(*
    This function block is responsible for printing the results of the assertions using the built-in
    ADSLOGSTR functionality provided by the Tc2_System library. This sends the result using ADS, which
    is consumed by the error list of Visual Studio.
*)
FUNCTION_BLOCK FB_AdsAssertMessageFormatter IMPLEMENTS I_AssertMessageFormatter

METHOD PUBLIC LogAssertFailure
VAR_INPUT
    Expected : T_MaxString;
    Actual : T_MaxString;
    Message : T_MaxString;
    TestInstancePath : T_MaxString;
END_VAR
VAR
    AdjustAssertFailureMessageToMaxAllowedLength : FB_AdjustAssertFailureMessageToMaxAllowedLength;
    TestInstancePathCleaned : T_MaxString;
    TestInstancePathFinal : T_MaxString;
    ReturnValue : DINT;
    TestInstancePathProcessed : T_MaxString;
    MessagePart2 : T_MaxString;
    MessagePart3 : T_MaxString;
    MessagePart4 : T_MaxString;
    MessageProcessed : T_MaxString;
    Length2 : INT;
    Length3 : INT;
    Length4 : INT;
    LengthTotal : INT;
END_VAR
VAR CONSTANT
    MESSAGE_FORMATTED_STRING_MAX_NUMBER_OF_CHARACTERS : INT := 252; // The maximum printed text length is 250. The '%s' placeholder will be replaced, therefore the limit to use in the check is 252.
    ACTEXP_MAX_NUMBER_OF_CHARACTERS : INT := 250;
    TOO_LONG : STRING := '...too long';
END_VAR
TestInstancePathCleaned := F_RemoveInstancePathAndProjectNameFromTestInstancePath(TestInstancePath);
TestInstancePathFinal := CONCAT(STR1 := 'FAILED TEST $'',
                                STR2 := TestInstancePathCleaned);
TestInstancePathFinal := CONCAT(STR1 := TestInstancePathFinal,
                                STR2 := '$'');

MessagePart2 := CONCAT(STR1 := 'EXP: ',
                       STR2 := Expected);
MessagePart3 := CONCAT(STR1 := 'ACT: ',
                       STR2 := Actual);
IF LEN(STR := Message) > 0 THEN
    MessagePart4 := ', MSG: %s';
    Length4 := LEN(STR := MessagePart4)
             + LEN(STR := Message);
END_IF

IF (GVL_Param_TcUnit.MultipleLinesPerAssertionMessage) THEN
    Length2 := LEN(MessagePart2);
    IF (Length2 > ACTEXP_MAX_NUMBER_OF_CHARACTERS) THEN
        MessagePart2 := LEFT(STR := MessagePart2,
                             SIZE := ACTEXP_MAX_NUMBER_OF_CHARACTERS - LEN(STR := TOO_LONG));
        MessagePart2 := CONCAT (STR1 := MessagePart2,
                                STR2 := TOO_LONG);
        Length2 := LEN(MessagePart2);
    END_IF
    
    Length3 := LEN(MessagePart3);
    IF (Length3 > ACTEXP_MAX_NUMBER_OF_CHARACTERS) THEN
        MessagePart3 := LEFT(STR := MessagePart3,
                             SIZE := ACTEXP_MAX_NUMBER_OF_CHARACTERS - LEN(STR := TOO_LONG));
        MessagePart3 := CONCAT (STR1 := MessagePart3,
                                STR2 := TOO_LONG);
        Length3 := LEN(MessagePart3);
    END_IF

    LengthTotal := LEN(TestInstancePathFinal) + 2 + Length2 + 2 + Length3 + Length4;
END_IF

IF (LengthTotal <= MESSAGE_FORMATTED_STRING_MAX_NUMBER_OF_CHARACTERS) THEN
    // If the message must be printed on a single line ("multiple lines" disabled), then LengthTotal is not calculated, so this path is executed.
    TestInstancePathFinal := CONCAT(STR1 := TestInstancePathFinal,
                                    STR2 := ', ');
    TestInstancePathFinal := CONCAT(STR1 := TestInstancePathFinal,
                                    STR2 := MessagePart2);
    
    TestInstancePathFinal := CONCAT(STR1 := TestInstancePathFinal,
                                    STR2 := ', ');
    TestInstancePathFinal := CONCAT(STR1 := TestInstancePathFinal,
                                    STR2 := MessagePart3);
    
    IF Length4 > 0 THEN
        TestInstancePathFinal := CONCAT(STR1 := TestInstancePathFinal,
                                        STR2 := MessagePart4);
    END_IF
    
    AdjustAssertFailureMessageToMaxAllowedLength(TestInstancePath := TestInstancePathFinal,
                                                 TestMessage := Message,
                                                 TestInstancePathProcessed => TestInstancePathProcessed,
                                                 TestMessageProcessed => MessageProcessed);
    
    GVL_TcUnit.AdsMessageQueue.WriteLog(MsgCtrlMask := ADSLOG_MSGTYPE_ERROR,
                                        MsgFmtStr := TestInstancePathProcessed,
                                        StrArg := MessageProcessed);
    
// ELSE: print multiple lines
ELSIF (LEN(TestInstancePathFinal) + 2 + Length2 + 2 + Length3 <= MESSAGE_FORMATTED_STRING_MAX_NUMBER_OF_CHARACTERS) THEN
    // A message exists, because the text with message does not fit in one line, but it fits without the message. Print only the message in a separate line.
    TestInstancePathFinal := CONCAT(STR1 := TestInstancePathFinal,
                                    STR2 := ', ');
    TestInstancePathFinal := CONCAT(STR1 := TestInstancePathFinal,
                                    STR2 := MessagePart2);
    
    TestInstancePathFinal := CONCAT(STR1 := TestInstancePathFinal,
                                    STR2 := ', ');
    TestInstancePathFinal := CONCAT(STR1 := TestInstancePathFinal,
                                    STR2 := MessagePart3);
    
    AdjustAssertFailureMessageToMaxAllowedLength(TestInstancePath := TestInstancePathFinal,
                                                 TestMessage := '',
                                                 TestInstancePathProcessed => TestInstancePathProcessed,
                                                 TestMessageProcessed => MessageProcessed);
    
    GVL_TcUnit.AdsMessageQueue.WriteLog(MsgCtrlMask := ADSLOG_MSGTYPE_ERROR,
                                        MsgFmtStr := TestInstancePathProcessed,
                                        StrArg := MessageProcessed);
    
    // MessagePart4 (MSG)
    AdjustAssertFailureMessageToMaxAllowedLength(TestInstancePath := '_ MSG: %s',
                                                 TestMessage := Message,
                                                 TestInstancePathProcessed => TestInstancePathProcessed,
                                                 TestMessageProcessed => MessageProcessed);
    
    GVL_TcUnit.AdsMessageQueue.WriteLog(MsgCtrlMask := ADSLOG_MSGTYPE_ERROR,
                                        MsgFmtStr := TestInstancePathProcessed,
                                        StrArg := MessageProcessed);
    
ELSIF (2 + Length2 + 2 + Length3 <= ACTEXP_MAX_NUMBER_OF_CHARACTERS) THEN
    // Text without message does not fit in one line. EXP and ACT fit in one line, therefore print them together in 2nd line. Print message (if existing) in 3rd line.
    AdjustAssertFailureMessageToMaxAllowedLength(TestInstancePath := TestInstancePathFinal,
                                                 TestMessage := '',
                                                 TestInstancePathProcessed => TestInstancePathProcessed,
                                                 TestMessageProcessed => MessageProcessed);
    
    GVL_TcUnit.AdsMessageQueue.WriteLog(MsgCtrlMask := ADSLOG_MSGTYPE_ERROR,
                                        MsgFmtStr := TestInstancePathProcessed,
                                        StrArg := MessageProcessed);
    
    // MessagePart2 (EXP) + MessagePart3 (ACT)
    MessagePart2 := CONCAT (STR1 := '_ ',
                            STR2 := MessagePart2);
    MessagePart2 := CONCAT (STR1 := MessagePart2,
                            STR2 := ', ');
    MessagePart2 := CONCAT (STR1 := MessagePart2,
                            STR2 := MessagePart3);
    
    AdjustAssertFailureMessageToMaxAllowedLength(TestInstancePath := MessagePart2,
                                                 TestMessage := '',
                                                 TestInstancePathProcessed => TestInstancePathProcessed,
                                                 TestMessageProcessed => MessageProcessed);
    
    GVL_TcUnit.AdsMessageQueue.WriteLog(MsgCtrlMask := ADSLOG_MSGTYPE_ERROR,
                                        MsgFmtStr := TestInstancePathProcessed,
                                        StrArg := MessageProcessed);
    
    // MessagePart4 (MSG)
    IF Length4 > 0 THEN
        AdjustAssertFailureMessageToMaxAllowedLength(TestInstancePath := '_ MSG: %s',
                                                     TestMessage := Message,
                                                     TestInstancePathProcessed => TestInstancePathProcessed,
                                                     TestMessageProcessed => MessageProcessed);
        
        GVL_TcUnit.AdsMessageQueue.WriteLog(MsgCtrlMask := ADSLOG_MSGTYPE_ERROR,
                                            MsgFmtStr := TestInstancePathProcessed,
                                            StrArg := MessageProcessed);
    END_IF
ELSE
    // print every item in a separate line.
    AdjustAssertFailureMessageToMaxAllowedLength(TestInstancePath := TestInstancePathFinal,
                                                 TestMessage := '',
                                                 TestInstancePathProcessed => TestInstancePathProcessed,
                                                 TestMessageProcessed => MessageProcessed);
    
    GVL_TcUnit.AdsMessageQueue.WriteLog(MsgCtrlMask := ADSLOG_MSGTYPE_ERROR,
                                        MsgFmtStr := TestInstancePathProcessed,
                                        StrArg := MessageProcessed);
    
    // MessagePart2 (EXP)
    MessagePart2 := CONCAT (STR1 := '_ ',
                            STR2 := MessagePart2);

    AdjustAssertFailureMessageToMaxAllowedLength(TestInstancePath := MessagePart2,
                                                 TestMessage := '',
                                                 TestInstancePathProcessed => TestInstancePathProcessed,
                                                 TestMessageProcessed => MessageProcessed);
    
    GVL_TcUnit.AdsMessageQueue.WriteLog(MsgCtrlMask := ADSLOG_MSGTYPE_ERROR,
                                        MsgFmtStr := TestInstancePathProcessed,
                                        StrArg := MessageProcessed);
    
    // MessagePart3 (ACT)
    MessagePart3 := CONCAT (STR1 := '_ ',
                            STR2 := MessagePart3);
    
    AdjustAssertFailureMessageToMaxAllowedLength(TestInstancePath := MessagePart3,
                                                 TestMessage := '',
                                                 TestInstancePathProcessed => TestInstancePathProcessed,
                                                 TestMessageProcessed => MessageProcessed);
    
    GVL_TcUnit.AdsMessageQueue.WriteLog(MsgCtrlMask := ADSLOG_MSGTYPE_ERROR,
                                        MsgFmtStr := TestInstancePathProcessed,
                                        StrArg := MessageProcessed);
    
    // MessagePart4 (MSG)
    IF Length4 > 0 THEN
        AdjustAssertFailureMessageToMaxAllowedLength(TestInstancePath := '_ MSG: %s',
                                                     TestMessage := Message,
                                                     TestInstancePathProcessed => TestInstancePathProcessed,
                                                     TestMessageProcessed => MessageProcessed);
        
        GVL_TcUnit.AdsMessageQueue.WriteLog(MsgCtrlMask := ADSLOG_MSGTYPE_ERROR,
                                            MsgFmtStr := TestInstancePathProcessed,
                                            StrArg := MessageProcessed);
    END_IF
END_IF
END_METHOD

END_FUNCTION_BLOCK

(* stored: Version 1.1.0.1
   POU FB_AdsAssertMessageFormatter: Id {54911d7d-b4a4-43a8-a981-a2fc14a13f71}, SpecialFunc None
   Method LogAssertFailure: Id {48cbc6b0-5380-44b8-a045-57b6ad9f189d} *)
